Staubli VAL3: onExit.pgx

program onExit(bool& x_bSave[])
  local string l_sMessage
  local bool l_bYes
  local bool l_bCancel
  local string l_sButton[2]
begin
  //
  // saveIt
  //
  if x_bSave
    call language:message(l_sMessage,-1)
    // get the yes_no button Key
    call language:getYesNo(l_sButton)
    // ask the question
    call use:yes_no_cancel(l_sMessage,l_sButton,l_bYes,l_bCancel)
    if l_bYes
      call saveIt(x_bSave)
    endIf
    // quit if not cancel
    bExit=!l_bCancel
  else
    // exit
    bExit=true
  endIf
end
